// TIA Portal V17 export
// export: Created 2025-03-13T10:30:57.8594611Z, ExportSetting WithDefaults, DisplayName Totally Integrated Automation Portal, DisplayVersion V17 Update 8, DisplayName TIA Portal Openness, DisplayVersion V17 Update 8, DisplayName TIA Portal Version Control Interface, DisplayVersion V17, DisplayName SINAMICS Startdrive Advanced, DisplayVersion V17 SP2, DisplayName SINAMICS Startdrive G110M, G120, G120C, G120D, G120P, G115D, DisplayVersion V17 SP2, DisplayName SINAMICS Startdrive G130, G150, S120, S150, SINAMICS MV, S210, DisplayVersion V17 SP2, DisplayName STEP 7 Professional, DisplayVersion V17 Update 8, DisplayName SINUMERIK ONE STEP 7 Toolbox, DisplayVersion V17 Update 12, DisplayName SINUMERIK 840D sl STEP 7 Toolbox, DisplayVersion V17 Update 12, DisplayName STEP 7 Safety, DisplayVersion V17 Update 6, DisplayName WinCC Advanced, DisplayVersion V17 Update 8
DATA_BLOCK "DB505_HMI_SetUp"   // DB505
{ S7_Optimized_Access := 'FALSE'; DB_Accessible_From_OPC_UA := 'FALSE' }
AUTHOR : ETXETAR
VERSION : 1.0
// stored: AutoNumber false, DBAccessibleFromOPCUA false, DBAccessibleFromWebserver true, IsOnlyStoredInLoadMemory false, IsWriteProtectedInAS false
   VAR
      Setup1 : Struct
         Movement_EndPos : Struct   // Movement End Pos
            movement1EndPosLeft : Bool;   // Movement End Pos
            movement1EndPosRight : Bool;   // Movement End Pos
            movement2EndPosLeft : Bool;   // Movement End Pos
            movement2EndPosRight : Bool;   // Movement End Pos
            movement3EndPosLeft : Bool;   // Movement End Pos
            movement3EndPosRight : Bool;   // Movement End Pos
            movement4EndPosLeft : Bool;   // Movement End Pos
            movement4EndPosRight : Bool;   // Movement End Pos
            movement5EndPosLeft : Bool;   // Movement End Pos
            movement5EndPosRight : Bool;   // Movement End Pos
            movement6EndPosLeft : Bool;   // Movement End Pos
            movement6EndPosRight : Bool;   // Movement End Pos
            movement7EndPosLeft : Bool;   // Movement End Pos
            movement7EndPosRight : Bool;   // Movement End Pos
            movement8EndPosLeft : Bool;   // Movement End Pos
            movement8EndPosRight : Bool;   // Movement End Pos
            movement9EndPosLeft : Bool;   // Movement End Pos
            movement9EndPosRight : Bool;   // Movement End Pos
            movement10EndPosLeft : Bool;   // Movement End Pos
            movement10EndPosRight : Bool;   // Movement End Pos
            movement11EndPosLeft : Bool;   // Movement End Pos
            movement11EndPosRight : Bool;   // Movement End Pos
            movement12EndPosLeft : Bool;   // Movement End Pos
            movement12EndPosRight : Bool;   // Movement End Pos
            movement13EndPosLeft : Bool;   // Movement End Pos
            movement13EndPosRight : Bool;   // Movement End Pos
            movement14EndPosLeft : Bool;   // Movement End Pos
            movement14EndPosRight : Bool;   // Movement End Pos
            movement15EndPosLeft : Bool;   // Movement End Pos
            movement15EndPosRight : Bool;   // Movement End Pos
            movement16EndPosLeft : Bool;   // Movement End Pos
            movement16EndPosRight : Bool;   // Movement End Pos
            movement17EndPosLeft : Bool;   // Movement End Pos
            movement17EndPosRight : Bool;   // Movement End Pos
            movement18EndPosLeft : Bool;   // Movement End Pos
            movement18EndPosRight : Bool;   // Movement End Pos
            movement19EndPosLeft : Bool;   // Movement End Pos
            movement19EndPosRight : Bool;   // Movement End Pos
            movement20EndPosLeft : Bool;   // Movement End Pos
            movement20EndPosRight : Bool;   // Movement End Pos
            movement21EndPosLeft : Bool;   // Movement End Pos
            movement21EndPosRight : Bool;   // Movement End Pos
            movement22EndPosLeft : Bool;   // Movement End Pos
            movement22EndPosRight : Bool;   // Movement End Pos
            movement23EndPosLeft : Bool;   // Movement End Pos
            movement23EndPosRight : Bool;   // Movement End Pos
            movement24EndPosLeft : Bool;   // Movement End Pos
            movement24EndPosRight : Bool;   // Movement End Pos
            movement25EndPosLeft : Bool;   // Movement End Pos
            movement25EndPosRight : Bool;   // Movement End Pos
            movement26EndPosLeft : Bool;   // Movement End Pos
            movement26EndPosRight : Bool;   // Movement End Pos
            movement27EndPosLeft : Bool;   // Movement End Pos
            movement27EndPosRight : Bool;   // Movement End Pos
            movement28EndPosLeft : Bool;   // Movement End Pos
            movement28EndPosRight : Bool;   // Movement End Pos
            movement29EndPosLeft : Bool;   // Movement End Pos
            movement29EndPosRight : Bool;   // Movement End Pos
            movement30EndPosLeft : Bool;   // Movement End Pos
            movement30EndPosRight : Bool;   // Movement End Pos
            movement31EndPosLeft : Bool;   // Movement End Pos
            movement31EndPosRight : Bool;   // Movement End Pos
            movement32EndPosLeft : Bool;   // Movement End Pos
            movement32EndPosRight : Bool;   // Movement End Pos
            movement33EndPosLeft : Bool;   // Movement End Pos
            movement33EndPosRight : Bool;   // Movement End Pos
            movement34EndPosLeft : Bool;   // Movement End Pos
            movement34EndPosRight : Bool;   // Movement End Pos
            movement35EndPosLeft : Bool;   // Movement End Pos
            movement35EndPosRight : Bool;   // Movement End Pos
            movement36EndPosLeft : Bool;   // Movement End Pos
            movement36EndPosRight : Bool;   // Movement End Pos
            movement37EndPosLeft : Bool;   // Movement End Pos
            movement37EndPosRight : Bool;   // Movement End Pos
            movement38EndPosLeft : Bool;   // Movement End Pos
            movement38EndPosRight : Bool;   // Movement End Pos
            movement39EndPosLeft : Bool;   // Movement End Pos
            movement39EndPosRight : Bool;   // Movement End Pos
            movement40EndPosLeft : Bool;   // Movement End Pos
            movement40EndPosRight : Bool;   // Movement End Pos
            movement41EndPosLeft : Bool;   // Movement End Pos
            movement41EndPosRight : Bool;   // Movement End Pos
            movement42EndPosLeft : Bool;   // Movement End Pos
            movement42EndPosRight : Bool;   // Movement End Pos
            movement43EndPosLeft : Bool;   // Movement End Pos
            movement43EndPosRight : Bool;   // Movement End Pos
            movement44EndPosLeft : Bool;   // Movement End Pos
            movement44EndPosRight : Bool;   // Movement End Pos
            movement45EndPosLeft : Bool;   // Movement End Pos
            movement45EndPosRight : Bool;   // Movement End Pos
            movement46EndPosLeft : Bool;   // Movement End Pos
            movement46EndPosRight : Bool;   // Movement End Pos
            movement47EndPosLeft : Bool;   // Movement End Pos
            movement47EndPosRight : Bool;   // Movement End Pos
            movement48EndPosLeft : Bool;   // Movement End Pos
            movement48EndPosRight : Bool;   // Movement End Pos
            movement49EndPosLeft : Bool;   // Movement End Pos
            movement49EndPosRight : Bool;   // Movement End Pos
            movement50EndPosLeft : Bool;   // Movement End Pos
            movement50EndPosRight : Bool;   // Movement End Pos
            movement51EndPosLeft : Bool;   // Movement End Pos
            movement51EndPosRight : Bool;   // Movement End Pos
            movement52EndPosLeft : Bool;   // Movement End Pos
            movement52EndPosRight : Bool;   // Movement End Pos
            movement53EndPosLeft : Bool;   // Movement End Pos
            movement53EndPosRight : Bool;   // Movement End Pos
            movement54EndPosLeft : Bool;   // Movement End Pos
            movement54EndPosRight : Bool;   // Movement End Pos
            movement55EndPosLeft : Bool;   // Movement End Pos
            movement55EndPosRight : Bool;   // Movement End Pos
            movement56EndPosLeft : Bool;   // Movement End Pos
            movement56EndPosRight : Bool;   // Movement End Pos
            movement57EndPosLeft : Bool;   // Movement End Pos
            movement57EndPosRight : Bool;   // Movement End Pos
            movement58EndPosLeft : Bool;   // Movement End Pos
            movement58EndPosRight : Bool;   // Movement End Pos
            movement59EndPosLeft : Bool;   // Movement End Pos
            movement59EndPosRight : Bool;   // Movement End Pos
            movement60EndPosLeft : Bool;   // Movement End Pos
            movement60EndPosRight : Bool;   // Movement End Pos
            movement61EndPosLeft : Bool;   // Movement End Pos
            movement61EndPosRight : Bool;   // Movement End Pos
            movement62EndPosLeft : Bool;   // Movement End Pos
            movement62EndPosRight : Bool;   // Movement End Pos
            movement63EndPosLeft : Bool;   // Movement End Pos
            movement63EndPosRight : Bool;   // Movement End Pos
            movement64EndPosLeft : Bool;   // Movement End Pos
            movement64EndPosRight : Bool;   // Movement End Pos
            movement65EndPosLeft : Bool;   // Movement End Pos
            movement65EndPosRight : Bool;   // Movement End Pos
            movement66EndPosLeft : Bool;   // Movement End Pos
            movement66EndPosRight : Bool;   // Movement End Pos
            movement67EndPosLeft : Bool;   // Movement End Pos
            movement67EndPosRight : Bool;   // Movement End Pos
            movement68EndPosLeft : Bool;   // Movement End Pos
            movement68EndPosRight : Bool;   // Movement End Pos
            movement69EndPosLeft : Bool;   // Movement End Pos
            movement69EndPosRight : Bool;   // Movement End Pos
            movement70EndPosLeft : Bool;   // Movement End Pos
            movement70EndPosRight : Bool;   // Movement End Pos
            movement71EndPosLeft : Bool;   // Movement End Pos
            movement71EndPosRight : Bool;   // Movement End Pos
            movement72EndPosLeft : Bool;   // Movement End Pos
            movement72EndPosRight : Bool;   // Movement End Pos
            movement73EndPosLeft : Bool;   // Movement End Pos
            movement73EndPosRight : Bool;   // Movement End Pos
            movement74EndPosLeft : Bool;   // Movement End Pos
            movement74EndPosRight : Bool;   // Movement End Pos
            movement75EndPosLeft : Bool;   // Movement End Pos
            movement75EndPosRight : Bool;   // Movement End Pos
            movement76EndPosLeft : Bool;   // Movement End Pos
            movement76EndPosRight : Bool;   // Movement End Pos
            movement77EndPosLeft : Bool;   // Movement End Pos
            movement77EndPosRight : Bool;   // Movement End Pos
            movement78EndPosLeft : Bool;   // Movement End Pos
            movement78EndPosRight : Bool;   // Movement End Pos
            movement79EndPosLeft : Bool;   // Movement End Pos
            movement79EndPosRight : Bool;   // Movement End Pos
            movement80EndPosLeft : Bool;   // Movement End Pos
            movement80EndPosRight : Bool;   // Movement End Pos
            movement81EndPosLeft : Bool;   // Movement End Pos
            movement81EndPosRight : Bool;   // Movement End Pos
            movement82EndPosLeft : Bool;   // Movement End Pos
            movement82EndPosRight : Bool;   // Movement End Pos
            movement83EndPosLeft : Bool;   // Movement End Pos
            movement83EndPosRight : Bool;   // Movement End Pos
            movement84EndPosLeft : Bool;   // Movement End Pos
            movement84EndPosRight : Bool;   // Movement End Pos
            movement85EndPosLeft : Bool;   // Movement End Pos
            movement85EndPosRight : Bool;   // Movement End Pos
            movement86EndPosLeft : Bool;   // Movement End Pos
            movement86EndPosRight : Bool;   // Movement End Pos
            movement87EndPosLeft : Bool;   // Movement End Pos
            movement87EndPosRight : Bool;   // Movement End Pos
            movement88EndPosLeft : Bool;   // Movement End Pos
            movement88EndPosRight : Bool;   // Movement End Pos
            movement89EndPosLeft : Bool;   // Movement End Pos
            movement89EndPosRight : Bool;   // Movement End Pos
            movement90EndPosLeft : Bool;   // Movement End Pos
            movement90EndPosRight : Bool;   // Movement End Pos
            movement91EndPosLeft : Bool;   // Movement End Pos
            movement91EndPosRight : Bool;   // Movement End Pos
            movement92EndPosLeft : Bool;   // Movement End Pos
            movement92EndPosRight : Bool;   // Movement End Pos
            movement93EndPosLeft : Bool;   // Movement End Pos
            movement93EndPosRight : Bool;   // Movement End Pos
            movement94EndPosLeft : Bool;   // Movement End Pos
            movement94EndPosRight : Bool;   // Movement End Pos
            movement95EndPosLeft : Bool;   // Movement End Pos
            movement95EndPosRight : Bool;   // Movement End Pos
            movement96EndPosLeft : Bool;   // Movement End Pos
            movement96EndPosRight : Bool;   // Movement End Pos
            movement97EndPosLeft : Bool;   // Movement End Pos
            movement97EndPosRight : Bool;   // Movement End Pos
            movement98EndPosLeft : Bool;   // Movement End Pos
            movement98EndPosRight : Bool;   // Movement End Pos
            movement99EndPosLeft : Bool;   // Movement End Pos
            movement99EndPosRight : Bool;   // Movement End Pos
            movement100EndPosLeft : Bool;   // Movement End Pos
            movement100EndPosRight : Bool;   // Movement End Pos
            movement101EndPosLeft : Bool;   // Movement End Pos
            movement101EndPosRight : Bool;   // Movement End Pos
            movement102EndPosLeft : Bool;   // Movement End Pos
            movement102EndPosRight : Bool;   // Movement End Pos
            movement103EndPosLeft : Bool;   // Movement End Pos
            movement103EndPosRight : Bool;   // Movement End Pos
            movement104EndPosLeft : Bool;   // Movement End Pos
            movement104EndPosRight : Bool;   // Movement End Pos
            movement105EndPosLeft : Bool;   // Movement End Pos
            movement105EndPosRight : Bool;   // Movement End Pos
            movement106EndPosLeft : Bool;   // Movement End Pos
            movement106EndPosRight : Bool;   // Movement End Pos
            movement107EndPosLeft : Bool;   // Movement End Pos
            movement107EndPosRight : Bool;   // Movement End Pos
            movement108EndPosLeft : Bool;   // Movement End Pos
            movement108EndPosRight : Bool;   // Movement End Pos
            movement109EndPosLeft : Bool;   // Movement End Pos
            movement109EndPosRight : Bool;   // Movement End Pos
            movement110EndPosLeft : Bool;   // Movement End Pos
            movement110EndPosRight : Bool;   // Movement End Pos
            movement111EndPosLeft : Bool;   // Movement End Pos
            movement111EndPosRight : Bool;   // Movement End Pos
            movement112EndPosLeft : Bool;   // Movement End Pos
            movement112EndPosRight : Bool;   // Movement End Pos
            movement113EndPosLeft : Bool;   // Movement End Pos
            movement113EndPosRight : Bool;   // Movement End Pos
            movement114EndPosLeft : Bool;   // Movement End Pos
            movement114EndPosRight : Bool;   // Movement End Pos
            movement115EndPosLeft : Bool;   // Movement End Pos
            movement115EndPosRight : Bool;   // Movement End Pos
            movement116EndPosLeft : Bool;   // Movement End Pos
            movement116EndPosRight : Bool;   // Movement End Pos
            movement117EndPosLeft : Bool;   // Movement End Pos
            movement117EndPosRight : Bool;   // Movement End Pos
            movement118EndPosLeft : Bool;   // Movement End Pos
            movement118EndPosRight : Bool;   // Movement End Pos
            movement119EndPosLeft : Bool;   // Movement End Pos
            movement119EndPosRight : Bool;   // Movement End Pos
            movement120EndPosLeft : Bool;   // Movement End Pos
            movement120EndPosRight : Bool;   // Movement End Pos
            movement121EndPosLeft : Bool;   // Movement End Pos
            movement121EndPosRight : Bool;   // Movement End Pos
            movement122EndPosLeft : Bool;   // Movement End Pos
            movement122EndPosRight : Bool;   // Movement End Pos
            movement123EndPosLeft : Bool;   // Movement End Pos
            movement123EndPosRight : Bool;   // Movement End Pos
            movement124EndPosLeft : Bool;   // Movement End Pos
            movement124EndPosRight : Bool;   // Movement End Pos
            movement125EndPosLeft : Bool;   // Movement End Pos
            movement125EndPosRight : Bool;   // Movement End Pos
            movement126EndPosLeft : Bool;   // Movement End Pos
            movement126EndPosRight : Bool;   // Movement End Pos
            movement127EndPosLeft : Bool;   // Movement End Pos
            movement127EndPosRight : Bool;   // Movement End Pos
            movement128EndPosLeft : Bool;   // Movement End Pos
            movement128EndPosRight : Bool;   // Movement End Pos
            movement129EndPosLeft : Bool;   // Movement End Pos
            movement129EndPosRight : Bool;   // Movement End Pos
            movement130EndPosLeft : Bool;   // Movement End Pos
            movement130EndPosRight : Bool;   // Movement End Pos
            movement131EndPosLeft : Bool;   // Movement End Pos
            movement131EndPosRight : Bool;   // Movement End Pos
            movement132EndPosLeft : Bool;   // Movement End Pos
            movement132EndPosRight : Bool;   // Movement End Pos
            movement133EndPosLeft : Bool;   // Movement End Pos
            movement133EndPosRight : Bool;   // Movement End Pos
            movement134EndPosLeft : Bool;   // Movement End Pos
            movement134EndPosRight : Bool;   // Movement End Pos
            movement135EndPosLeft : Bool;   // Movement End Pos
            movement135EndPosRight : Bool;   // Movement End Pos
            movement136EndPosLeft : Bool;   // Movement End Pos
            movement136EndPosRight : Bool;   // Movement End Pos
            movement137EndPosLeft : Bool;   // Movement End Pos
            movement137EndPosRight : Bool;   // Movement End Pos
            movement138EndPosLeft : Bool;   // Movement End Pos
            movement138EndPosRight : Bool;   // Movement End Pos
            movement139EndPosLeft : Bool;   // Movement End Pos
            movement139EndPosRight : Bool;   // Movement End Pos
            movement140EndPosLeft : Bool;   // Movement End Pos
            movement140EndPosRight : Bool;   // Movement End Pos
            movement141EndPosLeft : Bool;   // Movement End Pos
            movement141EndPosRight : Bool;   // Movement End Pos
            movement142EndPosLeft : Bool;   // Movement End Pos
            movement142EndPosRight : Bool;   // Movement End Pos
            movement143EndPosLeft : Bool;   // Movement End Pos
            movement143EndPosRight : Bool;   // Movement End Pos
            movement144EndPosLeft : Bool;   // Movement End Pos
            movement144EndPosRight : Bool;   // Movement End Pos
            movement145EndPosLeft : Bool;   // Movement End Pos
            movement145EndPosRight : Bool;   // Movement End Pos
            movement146EndPosLeft : Bool;   // Movement End Pos
            movement146EndPosRight : Bool;   // Movement End Pos
            movement147EndPosLeft : Bool;   // Movement End Pos
            movement147EndPosRight : Bool;   // Movement End Pos
            movement148EndPosLeft : Bool;   // Movement End Pos
            movement148EndPosRight : Bool;   // Movement End Pos
            movement149EndPosLeft : Bool;   // Movement End Pos
            movement149EndPosRight : Bool;   // Movement End Pos
            movement150EndPosLeft : Bool;   // Movement End Pos
            movement150EndPosRight : Bool;   // Movement End Pos
            movement151EndPosLeft : Bool;   // Movement End Pos
            movement151EndPosRight : Bool;   // Movement End Pos
            movement152EndPosLeft : Bool;   // Movement End Pos
            movement152EndPosRight : Bool;   // Movement End Pos
            movement153EndPosLeft : Bool;   // Movement End Pos
            movement153EndPosRight : Bool;   // Movement End Pos
            movement154EndPosLeft : Bool;   // Movement End Pos
            movement154EndPosRight : Bool;   // Movement End Pos
            movement155EndPosLeft : Bool;   // Movement End Pos
            movement155EndPosRight : Bool;   // Movement End Pos
            movement156EndPosLeft : Bool;   // Movement End Pos
            movement156EndPosRight : Bool;   // Movement End Pos
            movement157EndPosLeft : Bool;   // Movement End Pos
            movement157EndPosRight : Bool;   // Movement End Pos
            movement158EndPosLeft : Bool;   // Movement End Pos
            movement158EndPosRight : Bool;   // Movement End Pos
            movement159EndPosLeft : Bool;   // Movement End Pos
            movement159EndPosRight : Bool;   // Movement End Pos
            movement160EndPosLeft : Bool;   // Movement End Pos
            movement160EndPosRight : Bool;   // Movement End Pos
            movement161EndPosLeft : Bool;   // Movement End Pos
            movement161EndPosRight : Bool;   // Movement End Pos
            movement162EndPosLeft : Bool;   // Movement End Pos
            movement162EndPosRight : Bool;   // Movement End Pos
            movement163EndPosLeft : Bool;   // Movement End Pos
            movement163EndPosRight : Bool;   // Movement End Pos
            movement164EndPosLeft : Bool;   // Movement End Pos
            movement164EndPosRight : Bool;   // Movement End Pos
            movement165EndPosLeft : Bool;   // Movement End Pos
            movement165EndPosRight : Bool;   // Movement End Pos
            movement166EndPosLeft : Bool;   // Movement End Pos
            movement166EndPosRight : Bool;   // Movement End Pos
            movement167EndPosLeft : Bool;   // Movement End Pos
            movement167EndPosRight : Bool;   // Movement End Pos
            movement168EndPosLeft : Bool;   // Movement End Pos
            movement168EndPosRight : Bool;   // Movement End Pos
            movement169EndPosLeft : Bool;   // Movement End Pos
            movement169EndPosRight : Bool;   // Movement End Pos
            movement170EndPosLeft : Bool;   // Movement End Pos
            movement170EndPosRight : Bool;   // Movement End Pos
            movement171EndPosLeft : Bool;   // Movement End Pos
            movement171EndPosRight : Bool;   // Movement End Pos
            movement172EndPosLeft : Bool;   // Movement End Pos
            movement172EndPosRight : Bool;   // Movement End Pos
            movement173EndPosLeft : Bool;   // Movement End Pos
            movement173EndPosRight : Bool;   // Movement End Pos
            movement174EndPosLeft : Bool;   // Movement End Pos
            movement174EndPosRight : Bool;   // Movement End Pos
            movement175EndPosLeft : Bool;   // Movement End Pos
            movement175EndPosRight : Bool;   // Movement End Pos
            movement176EndPosLeft : Bool;   // Movement End Pos
            movement176EndPosRight : Bool;   // Movement End Pos
            movement177EndPosLeft : Bool;   // Movement End Pos
            movement177EndPosRight : Bool;   // Movement End Pos
            movement178EndPosLeft : Bool;   // Movement End Pos
            movement178EndPosRight : Bool;   // Movement End Pos
            movement179EndPosLeft : Bool;   // Movement End Pos
            movement179EndPosRight : Bool;   // Movement End Pos
            movement180EndPosLeft : Bool;   // Movement End Pos
            movement180EndPosRight : Bool;   // Movement End Pos
            movement181EndPosLeft : Bool;   // Movement End Pos
            movement181EndPosRight : Bool;   // Movement End Pos
            movement182EndPosLeft : Bool;   // Movement End Pos
            movement182EndPosRight : Bool;   // Movement End Pos
            movement183EndPosLeft : Bool;   // Movement End Pos
            movement183EndPosRight : Bool;   // Movement End Pos
            movement184EndPosLeft : Bool;   // Movement End Pos
            movement184EndPosRight : Bool;   // Movement End Pos
            movement185EndPosLeft : Bool;   // Movement End Pos
            movement185EndPosRight : Bool;   // Movement End Pos
            movement186EndPosLeft : Bool;   // Movement End Pos
            movement186EndPosRight : Bool;   // Movement End Pos
            movement187EndPosLeft : Bool;   // Movement End Pos
            movement187EndPosRight : Bool;   // Movement End Pos
            movement188EndPosLeft : Bool;   // Movement End Pos
            movement188EndPosRight : Bool;   // Movement End Pos
            movement189EndPosLeft : Bool;   // Movement End Pos
            movement189EndPosRight : Bool;   // Movement End Pos
            movement190EndPosLeft : Bool;   // Movement End Pos
            movement190EndPosRight : Bool;   // Movement End Pos
            movement191EndPosLeft : Bool;   // Movement End Pos
            movement191EndPosRight : Bool;   // Movement End Pos
            movement192EndPosLeft : Bool;   // Movement End Pos
            movement192EndPosRight : Bool;   // Movement End Pos
            movement193EndPosLeft : Bool;   // Movement End Pos
            movement193EndPosRight : Bool;   // Movement End Pos
            movement194EndPosLeft : Bool;   // Movement End Pos
            movement194EndPosRight : Bool;   // Movement End Pos
            movement195EndPosLeft : Bool;   // Movement End Pos
            movement195EndPosRight : Bool;   // Movement End Pos
            movement196EndPosLeft : Bool;   // Movement End Pos
            movement196EndPosRight : Bool;   // Movement End Pos
            movement197EndPosLeft : Bool;   // Movement End Pos
            movement197EndPosRight : Bool;   // Movement End Pos
            movement198EndPosLeft : Bool;   // Movement End Pos
            movement198EndPosRight : Bool;   // Movement End Pos
            movement199EndPosLeft : Bool;   // Movement End Pos
            movement199EndPosRight : Bool;   // Movement End Pos
            movement200EndPosLeft : Bool;   // Movement End Pos
            movement200EndPosRight : Bool;   // Movement End Pos
            movement201EndPosLeft : Bool;   // Movement End Pos
            movement201EndPosRight : Bool;   // Movement End Pos
            movement202EndPosLeft : Bool;   // Movement End Pos
            movement202EndPosRight : Bool;   // Movement End Pos
            movement203EndPosLeft : Bool;   // Movement End Pos
            movement203EndPosRight : Bool;   // Movement End Pos
            movement204EndPosLeft : Bool;   // Movement End Pos
            movement204EndPosRight : Bool;   // Movement End Pos
            movement205EndPosLeft : Bool;   // Movement End Pos
            movement205EndPosRight : Bool;   // Movement End Pos
            movement206EndPosLeft : Bool;   // Movement End Pos
            movement206EndPosRight : Bool;   // Movement End Pos
            movement207EndPosLeft : Bool;   // Movement End Pos
            movement207EndPosRight : Bool;   // Movement End Pos
            movement208EndPosLeft : Bool;   // Movement End Pos
            movement208EndPosRight : Bool;   // Movement End Pos
            movement209EndPosLeft : Bool;   // Movement End Pos
            movement209EndPosRight : Bool;   // Movement End Pos
            movement210EndPosLeft : Bool;   // Movement End Pos
            movement210EndPosRight : Bool;   // Movement End Pos
            movement211EndPosLeft : Bool;   // Movement End Pos
            movement211EndPosRight : Bool;   // Movement End Pos
            movement212EndPosLeft : Bool;   // Movement End Pos
            movement212EndPosRight : Bool;   // Movement End Pos
            movement213EndPosLeft : Bool;   // Movement End Pos
            movement213EndPosRight : Bool;   // Movement End Pos
            movement214EndPosLeft : Bool;   // Movement End Pos
            movement214EndPosRight : Bool;   // Movement End Pos
            movement215EndPosLeft : Bool;   // Movement End Pos
            movement215EndPosRight : Bool;   // Movement End Pos
            movement216EndPosLeft : Bool;   // Movement End Pos
            movement216EndPosRight : Bool;   // Movement End Pos
            movement217EndPosLeft : Bool;   // Movement End Pos
            movement217EndPosRight : Bool;   // Movement End Pos
            movement218EndPosLeft : Bool;   // Movement End Pos
            movement218EndPosRight : Bool;   // Movement End Pos
            movement219EndPosLeft : Bool;   // Movement End Pos
            movement219EndPosRight : Bool;   // Movement End Pos
            movement220EndPosLeft : Bool;   // Movement End Pos
            movement220EndPosRight : Bool;   // Movement End Pos
            movement221EndPosLeft : Bool;   // Movement End Pos
            movement221EndPosRight : Bool;   // Movement End Pos
            movement222EndPosLeft : Bool;   // Movement End Pos
            movement222EndPosRight : Bool;   // Movement End Pos
            movement223EndPosLeft : Bool;   // Movement End Pos
            movement223EndPosRight : Bool;   // Movement End Pos
            movement224EndPosLeft : Bool;   // Movement End Pos
            movement224EndPosRight : Bool;   // Movement End Pos
            movement225EndPosLeft : Bool;   // Movement End Pos
            movement225EndPosRight : Bool;   // Movement End Pos
            movement226EndPosLeft : Bool;   // Movement End Pos
            movement226EndPosRight : Bool;   // Movement End Pos
            movement227EndPosLeft : Bool;   // Movement End Pos
            movement227EndPosRight : Bool;   // Movement End Pos
            movement228EndPosLeft : Bool;   // Movement End Pos
            movement228EndPosRight : Bool;   // Movement End Pos
            movement229EndPosLeft : Bool;   // Movement End Pos
            movement229EndPosRight : Bool;   // Movement End Pos
            movement230EndPosLeft : Bool;   // Movement End Pos
            movement230EndPosRight : Bool;   // Movement End Pos
            movement231EndPosLeft : Bool;   // Movement End Pos
            movement231EndPosRight : Bool;   // Movement End Pos
            movement232EndPosLeft : Bool;   // Movement End Pos
            movement232EndPosRight : Bool;   // Movement End Pos
            movement233EndPosLeft : Bool;   // Movement End Pos
            movement233EndPosRight : Bool;   // Movement End Pos
            movement234EndPosLeft : Bool;   // Movement End Pos
            movement234EndPosRight : Bool;   // Movement End Pos
            movement235EndPosLeft : Bool;   // Movement End Pos
            movement235EndPosRight : Bool;   // Movement End Pos
            movement236EndPosLeft : Bool;   // Movement End Pos
            movement236EndPosRight : Bool;   // Movement End Pos
            movement237EndPosLeft : Bool;   // Movement End Pos
            movement237EndPosRight : Bool;   // Movement End Pos
            movement238EndPosLeft : Bool;   // Movement End Pos
            movement238EndPosRight : Bool;   // Movement End Pos
            movement239EndPosLeft : Bool;   // Movement End Pos
            movement239EndPosRight : Bool;   // Movement End Pos
            movement240EndPosLeft : Bool;   // Movement End Pos
            movement240EndPosRight : Bool;   // Movement End Pos
            movement241EndPosLeft : Bool;   // Movement End Pos
            movement241EndPosRight : Bool;   // Movement End Pos
            movement242EndPosLeft : Bool;   // Movement End Pos
            movement242EndPosRight : Bool;   // Movement End Pos
            movement243EndPosLeft : Bool;   // Movement End Pos
            movement243EndPosRight : Bool;   // Movement End Pos
            movement244EndPosLeft : Bool;   // Movement End Pos
            movement244EndPosRight : Bool;   // Movement End Pos
            movement245EndPosLeft : Bool;   // Movement End Pos
            movement245EndPosRight : Bool;   // Movement End Pos
            movement246EndPosLeft : Bool;   // Movement End Pos
            movement246EndPosRight : Bool;   // Movement End Pos
            movement247EndPosLeft : Bool;   // Movement End Pos
            movement247EndPosRight : Bool;   // Movement End Pos
            movement248EndPosLeft : Bool;   // Movement End Pos
            movement248EndPosRight : Bool;   // Movement End Pos
            movement249EndPosLeft : Bool;   // Movement End Pos
            movement249EndPosRight : Bool;   // Movement End Pos
            movement250EndPosLeft : Bool;   // Movement End Pos
            movement250EndPosRight : Bool;   // Movement End Pos
            movement251EndPosLeft : Bool;   // Movement End Pos
            movement251EndPosRight : Bool;   // Movement End Pos
            movement252EndPosLeft : Bool;   // Movement End Pos
            movement252EndPosRight : Bool;   // Movement End Pos
            movement253EndPosLeft : Bool;   // Movement End Pos
            movement253EndPosRight : Bool;   // Movement End Pos
            movement254EndPosLeft : Bool;   // Movement End Pos
            movement254EndPosRight : Bool;   // Movement End Pos
            movement255EndPosLeft : Bool;   // Movement End Pos
            movement255EndPosRight : Bool;   // Movement End Pos
            movement256EndPosLeft : Bool;   // Movement End Pos
            movement256EndPosRight : Bool;   // Movement End Pos
         END_STRUCT;
         Movement_Executability : Struct   // Movement Executability
            movement1ExecutabilityLeft : Bool;   // Movement Executability
            movement1ExecutabilityRight : Bool;   // Movement Executability
            movement2ExecutabilityLeft : Bool;   // Movement Executability
            movement2ExecutabilityRight : Bool;   // Movement Executability
            movement3ExecutabilityLeft : Bool;   // Movement Executability
            movement3ExecutabilityRight : Bool;   // Movement Executability
            movement4ExecutabilityLeft : Bool;   // Movement Executability
            movement4ExecutabilityRight : Bool;   // Movement Executability
            movement5ExecutabilityLeft : Bool;   // Movement Executability
            movement5ExecutabilityRight : Bool;   // Movement Executability
            movement6ExecutabilityLeft : Bool;   // Movement Executability
            movement6ExecutabilityRight : Bool;   // Movement Executability
            movement7ExecutabilityLeft : Bool;   // Movement Executability
            movement7ExecutabilityRight : Bool;   // Movement Executability
            movement8ExecutabilityLeft : Bool;   // Movement Executability
            movement8ExecutabilityRight : Bool;   // Movement Executability
            movement9ExecutabilityLeft : Bool;   // Movement Executability
            movement9ExecutabilityRight : Bool;   // Movement Executability
            movement10ExecutabilityLeft : Bool;   // Movement Executability
            movement10ExecutabilityRight : Bool;   // Movement Executability
            movement11ExecutabilityLeft : Bool;   // Movement Executability
            movement11ExecutabilityRight : Bool;   // Movement Executability
            movement12ExecutabilityLeft : Bool;   // Movement Executability
            movement12ExecutabilityRight : Bool;   // Movement Executability
            movement13ExecutabilityLeft : Bool;   // Movement Executability
            movement13ExecutabilityRight : Bool;   // Movement Executability
            movement14ExecutabilityLeft : Bool;   // Movement Executability
            movement14ExecutabilityRight : Bool;   // Movement Executability
            movement15ExecutabilityLeft : Bool;   // Movement Executability
            movement15ExecutabilityRight : Bool;   // Movement Executability
            movement16ExecutabilityLeft : Bool;   // Movement Executability
            movement16ExecutabilityRight : Bool;   // Movement Executability
            movement17ExecutabilityLeft : Bool;   // Movement Executability
            movement17ExecutabilityRight : Bool;   // Movement Executability
            movement18ExecutabilityLeft : Bool;   // Movement Executability
            movement18ExecutabilityRight : Bool;   // Movement Executability
            movement19ExecutabilityLeft : Bool;   // Movement Executability
            movement19ExecutabilityRight : Bool;   // Movement Executability
            movement20ExecutabilityLeft : Bool;   // Movement Executability
            movement20ExecutabilityRight : Bool;   // Movement Executability
            movement21ExecutabilityLeft : Bool;   // Movement Executability
            movement21ExecutabilityRight : Bool;   // Movement Executability
            movement22ExecutabilityLeft : Bool;   // Movement Executability
            movement22ExecutabilityRight : Bool;   // Movement Executability
            movement23ExecutabilityLeft : Bool;   // Movement Executability
            movement23ExecutabilityRight : Bool;   // Movement Executability
            movement24ExecutabilityLeft : Bool;   // Movement Executability
            movement24ExecutabilityRight : Bool;   // Movement Executability
            movement25ExecutabilityLeft : Bool;   // Movement Executability
            movement25ExecutabilityRight : Bool;   // Movement Executability
            movement26ExecutabilityLeft : Bool;   // Movement Executability
            movement26ExecutabilityRight : Bool;   // Movement Executability
            movement27ExecutabilityLeft : Bool;   // Movement Executability
            movement27ExecutabilityRight : Bool;   // Movement Executability
            movement28ExecutabilityLeft : Bool;   // Movement Executability
            movement28ExecutabilityRight : Bool;   // Movement Executability
            movement29ExecutabilityLeft : Bool;   // Movement Executability
            movement29ExecutabilityRight : Bool;   // Movement Executability
            movement30ExecutabilityLeft : Bool;   // Movement Executability
            movement30ExecutabilityRight : Bool;   // Movement Executability
            movement31ExecutabilityLeft : Bool;   // Movement Executability
            movement31ExecutabilityRight : Bool;   // Movement Executability
            movement32ExecutabilityLeft : Bool;   // Movement Executability
            movement32ExecutabilityRight : Bool;   // Movement Executability
            movement33ExecutabilityLeft : Bool;   // Movement Executability
            movement33ExecutabilityRight : Bool;   // Movement Executability
            movement34ExecutabilityLeft : Bool;   // Movement Executability
            movement34ExecutabilityRight : Bool;   // Movement Executability
            movement35ExecutabilityLeft : Bool;   // Movement Executability
            movement35ExecutabilityRight : Bool;   // Movement Executability
            movement36ExecutabilityLeft : Bool;   // Movement Executability
            movement36ExecutabilityRight : Bool;   // Movement Executability
            movement37ExecutabilityLeft : Bool;   // Movement Executability
            movement37ExecutabilityRight : Bool;   // Movement Executability
            movement38ExecutabilityLeft : Bool;   // Movement Executability
            movement38ExecutabilityRight : Bool;   // Movement Executability
            movement39ExecutabilityLeft : Bool;   // Movement Executability
            movement39ExecutabilityRight : Bool;   // Movement Executability
            movement40ExecutabilityLeft : Bool;   // Movement Executability
            movement40ExecutabilityRight : Bool;   // Movement Executability
            movement41ExecutabilityLeft : Bool;   // Movement Executability
            movement41ExecutabilityRight : Bool;   // Movement Executability
            movement42ExecutabilityLeft : Bool;   // Movement Executability
            movement42ExecutabilityRight : Bool;   // Movement Executability
            movement43ExecutabilityLeft : Bool;   // Movement Executability
            movement43ExecutabilityRight : Bool;   // Movement Executability
            movement44ExecutabilityLeft : Bool;   // Movement Executability
            movement44ExecutabilityRight : Bool;   // Movement Executability
            movement45ExecutabilityLeft : Bool;   // Movement Executability
            movement45ExecutabilityRight : Bool;   // Movement Executability
            movement46ExecutabilityLeft : Bool;   // Movement Executability
            movement46ExecutabilityRight : Bool;   // Movement Executability
            movement47ExecutabilityLeft : Bool;   // Movement Executability
            movement47ExecutabilityRight : Bool;   // Movement Executability
            movement48ExecutabilityLeft : Bool;   // Movement Executability
            movement48ExecutabilityRight : Bool;   // Movement Executability
            movement49ExecutabilityLeft : Bool;   // Movement Executability
            movement49ExecutabilityRight : Bool;   // Movement Executability
            movement50ExecutabilityLeft : Bool;   // Movement Executability
            movement50ExecutabilityRight : Bool;   // Movement Executability
            movement51ExecutabilityLeft : Bool;   // Movement Executability
            movement51ExecutabilityRight : Bool;   // Movement Executability
            movement52ExecutabilityLeft : Bool;   // Movement Executability
            movement52ExecutabilityRight : Bool;   // Movement Executability
            movement53ExecutabilityLeft : Bool;   // Movement Executability
            movement53ExecutabilityRight : Bool;   // Movement Executability
            movement54ExecutabilityLeft : Bool;   // Movement Executability
            movement54ExecutabilityRight : Bool;   // Movement Executability
            movement55ExecutabilityLeft : Bool;   // Movement Executability
            movement55ExecutabilityRight : Bool;   // Movement Executability
            movement56ExecutabilityLeft : Bool;   // Movement Executability
            movement56ExecutabilityRight : Bool;   // Movement Executability
            movement57ExecutabilityLeft : Bool;   // Movement Executability
            movement57ExecutabilityRight : Bool;   // Movement Executability
            movement58ExecutabilityLeft : Bool;   // Movement Executability
            movement58ExecutabilityRight : Bool;   // Movement Executability
            movement59ExecutabilityLeft : Bool;   // Movement Executability
            movement59ExecutabilityRight : Bool;   // Movement Executability
            movement60ExecutabilityLeft : Bool;   // Movement Executability
            movement60ExecutabilityRight : Bool;   // Movement Executability
            movement61ExecutabilityLeft : Bool;   // Movement Executability
            movement61ExecutabilityRight : Bool;   // Movement Executability
            movement62ExecutabilityLeft : Bool;   // Movement Executability
            movement62ExecutabilityRight : Bool;   // Movement Executability
            movement63ExecutabilityLeft : Bool;   // Movement Executability
            movement63ExecutabilityRight : Bool;   // Movement Executability
            movement64ExecutabilityLeft : Bool;   // Movement Executability
            movement64ExecutabilityRight : Bool;   // Movement Executability
            movement65ExecutabilityLeft : Bool;   // Movement Executability
            movement65ExecutabilityRight : Bool;   // Movement Executability
            movement66ExecutabilityLeft : Bool;   // Movement Executability
            movement66ExecutabilityRight : Bool;   // Movement Executability
            movement67ExecutabilityLeft : Bool;   // Movement Executability
            movement67ExecutabilityRight : Bool;   // Movement Executability
            movement68ExecutabilityLeft : Bool;   // Movement Executability
            movement68ExecutabilityRight : Bool;   // Movement Executability
            movement69ExecutabilityLeft : Bool;   // Movement Executability
            movement69ExecutabilityRight : Bool;   // Movement Executability
            movement70ExecutabilityLeft : Bool;   // Movement Executability
            movement70ExecutabilityRight : Bool;   // Movement Executability
            movement71ExecutabilityLeft : Bool;   // Movement Executability
            movement71ExecutabilityRight : Bool;   // Movement Executability
            movement72ExecutabilityLeft : Bool;   // Movement Executability
            movement72ExecutabilityRight : Bool;   // Movement Executability
            movement73ExecutabilityLeft : Bool;   // Movement Executability
            movement73ExecutabilityRight : Bool;   // Movement Executability
            movement74ExecutabilityLeft : Bool;   // Movement Executability
            movement74ExecutabilityRight : Bool;   // Movement Executability
            movement75ExecutabilityLeft : Bool;   // Movement Executability
            movement75ExecutabilityRight : Bool;   // Movement Executability
            movement76ExecutabilityLeft : Bool;   // Movement Executability
            movement76ExecutabilityRight : Bool;   // Movement Executability
            movement77ExecutabilityLeft : Bool;   // Movement Executability
            movement77ExecutabilityRight : Bool;   // Movement Executability
            movement78ExecutabilityLeft : Bool;   // Movement Executability
            movement78ExecutabilityRight : Bool;   // Movement Executability
            movement79ExecutabilityLeft : Bool;   // Movement Executability
            movement79ExecutabilityRight : Bool;   // Movement Executability
            movement80ExecutabilityLeft : Bool;   // Movement Executability
            movement80ExecutabilityRight : Bool;   // Movement Executability
            movement81ExecutabilityLeft : Bool;   // Movement Executability
            movement81ExecutabilityRight : Bool;   // Movement Executability
            movement82ExecutabilityLeft : Bool;   // Movement Executability
            movement82ExecutabilityRight : Bool;   // Movement Executability
            movement83ExecutabilityLeft : Bool;   // Movement Executability
            movement83ExecutabilityRight : Bool;   // Movement Executability
            movement84ExecutabilityLeft : Bool;   // Movement Executability
            movement84ExecutabilityRight : Bool;   // Movement Executability
            movement85ExecutabilityLeft : Bool;   // Movement Executability
            movement85ExecutabilityRight : Bool;   // Movement Executability
            movement86ExecutabilityLeft : Bool;   // Movement Executability
            movement86ExecutabilityRight : Bool;   // Movement Executability
            movement87ExecutabilityLeft : Bool;   // Movement Executability
            movement87ExecutabilityRight : Bool;   // Movement Executability
            movement88ExecutabilityLeft : Bool;   // Movement Executability
            movement88ExecutabilityRight : Bool;   // Movement Executability
            movement89ExecutabilityLeft : Bool;   // Movement Executability
            movement89ExecutabilityRight : Bool;   // Movement Executability
            movement90ExecutabilityLeft : Bool;   // Movement Executability
            movement90ExecutabilityRight : Bool;   // Movement Executability
            movement91ExecutabilityLeft : Bool;   // Movement Executability
            movement91ExecutabilityRight : Bool;   // Movement Executability
            movement92ExecutabilityLeft : Bool;   // Movement Executability
            movement92ExecutabilityRight : Bool;   // Movement Executability
            movement93ExecutabilityLeft : Bool;   // Movement Executability
            movement93ExecutabilityRight : Bool;   // Movement Executability
            movement94ExecutabilityLeft : Bool;   // Movement Executability
            movement94ExecutabilityRight : Bool;   // Movement Executability
            movement95ExecutabilityLeft : Bool;   // Movement Executability
            movement95ExecutabilityRight : Bool;   // Movement Executability
            movement96ExecutabilityLeft : Bool;   // Movement Executability
            movement96ExecutabilityRight : Bool;   // Movement Executability
            movement97ExecutabilityLeft : Bool;   // Movement Executability
            movement97ExecutabilityRight : Bool;   // Movement Executability
            movement98ExecutabilityLeft : Bool;   // Movement Executability
            movement98ExecutabilityRight : Bool;   // Movement Executability
            movement99ExecutabilityLeft : Bool;   // Movement Executability
            movement99ExecutabilityRight : Bool;   // Movement Executability
            movement100ExecutabilityLeft : Bool;   // Movement Executability
            movement100ExecutabilityRight : Bool;   // Movement Executability
            movement101ExecutabilityLeft : Bool;   // Movement Executability
            movement101ExecutabilityRight : Bool;   // Movement Executability
            movement102ExecutabilityLeft : Bool;   // Movement Executability
            movement102ExecutabilityRight : Bool;   // Movement Executability
            movement103ExecutabilityLeft : Bool;   // Movement Executability
            movement103ExecutabilityRight : Bool;   // Movement Executability
            movement104ExecutabilityLeft : Bool;   // Movement Executability
            movement104ExecutabilityRight : Bool;   // Movement Executability
            movement105ExecutabilityLeft : Bool;   // Movement Executability
            movement105ExecutabilityRight : Bool;   // Movement Executability
            movement106ExecutabilityLeft : Bool;   // Movement Executability
            movement106ExecutabilityRight : Bool;   // Movement Executability
            movement107ExecutabilityLeft : Bool;   // Movement Executability
            movement107ExecutabilityRight : Bool;   // Movement Executability
            movement108ExecutabilityLeft : Bool;   // Movement Executability
            movement108ExecutabilityRight : Bool;   // Movement Executability
            movement109ExecutabilityLeft : Bool;   // Movement Executability
            movement109ExecutabilityRight : Bool;   // Movement Executability
            movement110ExecutabilityLeft : Bool;   // Movement Executability
            movement110ExecutabilityRight : Bool;   // Movement Executability
            movement111ExecutabilityLeft : Bool;   // Movement Executability
            movement111ExecutabilityRight : Bool;   // Movement Executability
            movement112ExecutabilityLeft : Bool;   // Movement Executability
            movement112ExecutabilityRight : Bool;   // Movement Executability
            movement113ExecutabilityLeft : Bool;   // Movement Executability
            movement113ExecutabilityRight : Bool;   // Movement Executability
            movement114ExecutabilityLeft : Bool;   // Movement Executability
            movement114ExecutabilityRight : Bool;   // Movement Executability
            movement115ExecutabilityLeft : Bool;   // Movement Executability
            movement115ExecutabilityRight : Bool;   // Movement Executability
            movement116ExecutabilityLeft : Bool;   // Movement Executability
            movement116ExecutabilityRight : Bool;   // Movement Executability
            movement117ExecutabilityLeft : Bool;   // Movement Executability
            movement117ExecutabilityRight : Bool;   // Movement Executability
            movement118ExecutabilityLeft : Bool;   // Movement Executability
            movement118ExecutabilityRight : Bool;   // Movement Executability
            movement119ExecutabilityLeft : Bool;   // Movement Executability
            movement119ExecutabilityRight : Bool;   // Movement Executability
            movement120ExecutabilityLeft : Bool;   // Movement Executability
            movement120ExecutabilityRight : Bool;   // Movement Executability
            movement121ExecutabilityLeft : Bool;   // Movement Executability
            movement121ExecutabilityRight : Bool;   // Movement Executability
            movement122ExecutabilityLeft : Bool;   // Movement Executability
            movement122ExecutabilityRight : Bool;   // Movement Executability
            movement123ExecutabilityLeft : Bool;   // Movement Executability
            movement123ExecutabilityRight : Bool;   // Movement Executability
            movement124ExecutabilityLeft : Bool;   // Movement Executability
            movement124ExecutabilityRight : Bool;   // Movement Executability
            movement125ExecutabilityLeft : Bool;   // Movement Executability
            movement125ExecutabilityRight : Bool;   // Movement Executability
            movement126ExecutabilityLeft : Bool;   // Movement Executability
            movement126ExecutabilityRight : Bool;   // Movement Executability
            movement127ExecutabilityLeft : Bool;   // Movement Executability
            movement127ExecutabilityRight : Bool;   // Movement Executability
            movement128ExecutabilityLeft : Bool;   // Movement Executability
            movement128ExecutabilityRight : Bool;   // Movement Executability
            movement129ExecutabilityLeft : Bool;   // Movement Executability
            movement129ExecutabilityRight : Bool;   // Movement Executability
            movement130ExecutabilityLeft : Bool;   // Movement Executability
            movement130ExecutabilityRight : Bool;   // Movement Executability
            movement131ExecutabilityLeft : Bool;   // Movement Executability
            movement131ExecutabilityRight : Bool;   // Movement Executability
            movement132ExecutabilityLeft : Bool;   // Movement Executability
            movement132ExecutabilityRight : Bool;   // Movement Executability
            movement133ExecutabilityLeft : Bool;   // Movement Executability
            movement133ExecutabilityRight : Bool;   // Movement Executability
            movement134ExecutabilityLeft : Bool;   // Movement Executability
            movement134ExecutabilityRight : Bool;   // Movement Executability
            movement135ExecutabilityLeft : Bool;   // Movement Executability
            movement135ExecutabilityRight : Bool;   // Movement Executability
            movement136ExecutabilityLeft : Bool;   // Movement Executability
            movement136ExecutabilityRight : Bool;   // Movement Executability
            movement137ExecutabilityLeft : Bool;   // Movement Executability
            movement137ExecutabilityRight : Bool;   // Movement Executability
            movement138ExecutabilityLeft : Bool;   // Movement Executability
            movement138ExecutabilityRight : Bool;   // Movement Executability
            movement139ExecutabilityLeft : Bool;   // Movement Executability
            movement139ExecutabilityRight : Bool;   // Movement Executability
            movement140ExecutabilityLeft : Bool;   // Movement Executability
            movement140ExecutabilityRight : Bool;   // Movement Executability
            movement141ExecutabilityLeft : Bool;   // Movement Executability
            movement141ExecutabilityRight : Bool;   // Movement Executability
            movement142ExecutabilityLeft : Bool;   // Movement Executability
            movement142ExecutabilityRight : Bool;   // Movement Executability
            movement143ExecutabilityLeft : Bool;   // Movement Executability
            movement143ExecutabilityRight : Bool;   // Movement Executability
            movement144ExecutabilityLeft : Bool;   // Movement Executability
            movement144ExecutabilityRight : Bool;   // Movement Executability
            movement145ExecutabilityLeft : Bool;   // Movement Executability
            movement145ExecutabilityRight : Bool;   // Movement Executability
            movement146ExecutabilityLeft : Bool;   // Movement Executability
            movement146ExecutabilityRight : Bool;   // Movement Executability
            movement147ExecutabilityLeft : Bool;   // Movement Executability
            movement147ExecutabilityRight : Bool;   // Movement Executability
            movement148ExecutabilityLeft : Bool;   // Movement Executability
            movement148ExecutabilityRight : Bool;   // Movement Executability
            movement149ExecutabilityLeft : Bool;   // Movement Executability
            movement149ExecutabilityRight : Bool;   // Movement Executability
            movement150ExecutabilityLeft : Bool;   // Movement Executability
            movement150ExecutabilityRight : Bool;   // Movement Executability
            movement151ExecutabilityLeft : Bool;   // Movement Executability
            movement151ExecutabilityRight : Bool;   // Movement Executability
            movement152ExecutabilityLeft : Bool;   // Movement Executability
            movement152ExecutabilityRight : Bool;   // Movement Executability
            movement153ExecutabilityLeft : Bool;   // Movement Executability
            movement153ExecutabilityRight : Bool;   // Movement Executability
            movement154ExecutabilityLeft : Bool;   // Movement Executability
            movement154ExecutabilityRight : Bool;   // Movement Executability
            movement155ExecutabilityLeft : Bool;   // Movement Executability
            movement155ExecutabilityRight : Bool;   // Movement Executability
            movement156ExecutabilityLeft : Bool;   // Movement Executability
            movement156ExecutabilityRight : Bool;   // Movement Executability
            movement157ExecutabilityLeft : Bool;   // Movement Executability
            movement157ExecutabilityRight : Bool;   // Movement Executability
            movement158ExecutabilityLeft : Bool;   // Movement Executability
            movement158ExecutabilityRight : Bool;   // Movement Executability
            movement159ExecutabilityLeft : Bool;   // Movement Executability
            movement159ExecutabilityRight : Bool;   // Movement Executability
            movement160ExecutabilityLeft : Bool;   // Movement Executability
            movement160ExecutabilityRight : Bool;   // Movement Executability
            movement161ExecutabilityLeft : Bool;   // Movement Executability
            movement161ExecutabilityRight : Bool;   // Movement Executability
            movement162ExecutabilityLeft : Bool;   // Movement Executability
            movement162ExecutabilityRight : Bool;   // Movement Executability
            movement163ExecutabilityLeft : Bool;   // Movement Executability
            movement163ExecutabilityRight : Bool;   // Movement Executability
            movement164ExecutabilityLeft : Bool;   // Movement Executability
            movement164ExecutabilityRight : Bool;   // Movement Executability
            movement165ExecutabilityLeft : Bool;   // Movement Executability
            movement165ExecutabilityRight : Bool;   // Movement Executability
            movement166ExecutabilityLeft : Bool;   // Movement Executability
            movement166ExecutabilityRight : Bool;   // Movement Executability
            movement167ExecutabilityLeft : Bool;   // Movement Executability
            movement167ExecutabilityRight : Bool;   // Movement Executability
            movement168ExecutabilityLeft : Bool;   // Movement Executability
            movement168ExecutabilityRight : Bool;   // Movement Executability
            movement169ExecutabilityLeft : Bool;   // Movement Executability
            movement169ExecutabilityRight : Bool;   // Movement Executability
            movement170ExecutabilityLeft : Bool;   // Movement Executability
            movement170ExecutabilityRight : Bool;   // Movement Executability
            movement171ExecutabilityLeft : Bool;   // Movement Executability
            movement171ExecutabilityRight : Bool;   // Movement Executability
            movement172ExecutabilityLeft : Bool;   // Movement Executability
            movement172ExecutabilityRight : Bool;   // Movement Executability
            movement173ExecutabilityLeft : Bool;   // Movement Executability
            movement173ExecutabilityRight : Bool;   // Movement Executability
            movement174ExecutabilityLeft : Bool;   // Movement Executability
            movement174ExecutabilityRight : Bool;   // Movement Executability
            movement175ExecutabilityLeft : Bool;   // Movement Executability
            movement175ExecutabilityRight : Bool;   // Movement Executability
            movement176ExecutabilityLeft : Bool;   // Movement Executability
            movement176ExecutabilityRight : Bool;   // Movement Executability
            movement177ExecutabilityLeft : Bool;   // Movement Executability
            movement177ExecutabilityRight : Bool;   // Movement Executability
            movement178ExecutabilityLeft : Bool;   // Movement Executability
            movement178ExecutabilityRight : Bool;   // Movement Executability
            movement179ExecutabilityLeft : Bool;   // Movement Executability
            movement179ExecutabilityRight : Bool;   // Movement Executability
            movement180ExecutabilityLeft : Bool;   // Movement Executability
            movement180ExecutabilityRight : Bool;   // Movement Executability
            movement181ExecutabilityLeft : Bool;   // Movement Executability
            movement181ExecutabilityRight : Bool;   // Movement Executability
            movement182ExecutabilityLeft : Bool;   // Movement Executability
            movement182ExecutabilityRight : Bool;   // Movement Executability
            movement183ExecutabilityLeft : Bool;   // Movement Executability
            movement183ExecutabilityRight : Bool;   // Movement Executability
            movement184ExecutabilityLeft : Bool;   // Movement Executability
            movement184ExecutabilityRight : Bool;   // Movement Executability
            movement185ExecutabilityLeft : Bool;   // Movement Executability
            movement185ExecutabilityRight : Bool;   // Movement Executability
            movement186ExecutabilityLeft : Bool;   // Movement Executability
            movement186ExecutabilityRight : Bool;   // Movement Executability
            movement187ExecutabilityLeft : Bool;   // Movement Executability
            movement187ExecutabilityRight : Bool;   // Movement Executability
            movement188ExecutabilityLeft : Bool;   // Movement Executability
            movement188ExecutabilityRight : Bool;   // Movement Executability
            movement189ExecutabilityLeft : Bool;   // Movement Executability
            movement189ExecutabilityRight : Bool;   // Movement Executability
            movement190ExecutabilityLeft : Bool;   // Movement Executability
            movement190ExecutabilityRight : Bool;   // Movement Executability
            movement191ExecutabilityLeft : Bool;   // Movement Executability
            movement191ExecutabilityRight : Bool;   // Movement Executability
            movement192ExecutabilityLeft : Bool;   // Movement Executability
            movement192ExecutabilityRight : Bool;   // Movement Executability
            movement193ExecutabilityLeft : Bool;   // Movement Executability
            movement193ExecutabilityRight : Bool;   // Movement Executability
            movement194ExecutabilityLeft : Bool;   // Movement Executability
            movement194ExecutabilityRight : Bool;   // Movement Executability
            movement195ExecutabilityLeft : Bool;   // Movement Executability
            movement195ExecutabilityRight : Bool;   // Movement Executability
            movement196ExecutabilityLeft : Bool;   // Movement Executability
            movement196ExecutabilityRight : Bool;   // Movement Executability
            movement197ExecutabilityLeft : Bool;   // Movement Executability
            movement197ExecutabilityRight : Bool;   // Movement Executability
            movement198ExecutabilityLeft : Bool;   // Movement Executability
            movement198ExecutabilityRight : Bool;   // Movement Executability
            movement199ExecutabilityLeft : Bool;   // Movement Executability
            movement199ExecutabilityRight : Bool;   // Movement Executability
            movement200ExecutabilityLeft : Bool;   // Movement Executability
            movement200ExecutabilityRight : Bool;   // Movement Executability
            movement201ExecutabilityLeft : Bool;   // Movement Executability
            movement201ExecutabilityRight : Bool;   // Movement Executability
            movement202ExecutabilityLeft : Bool;   // Movement Executability
            movement202ExecutabilityRight : Bool;   // Movement Executability
            movement203ExecutabilityLeft : Bool;   // Movement Executability
            movement203ExecutabilityRight : Bool;   // Movement Executability
            movement204ExecutabilityLeft : Bool;   // Movement Executability
            movement204ExecutabilityRight : Bool;   // Movement Executability
            movement205ExecutabilityLeft : Bool;   // Movement Executability
            movement205ExecutabilityRight : Bool;   // Movement Executability
            movement206ExecutabilityLeft : Bool;   // Movement Executability
            movement206ExecutabilityRight : Bool;   // Movement Executability
            movement207ExecutabilityLeft : Bool;   // Movement Executability
            movement207ExecutabilityRight : Bool;   // Movement Executability
            movement208ExecutabilityLeft : Bool;   // Movement Executability
            movement208ExecutabilityRight : Bool;   // Movement Executability
            movement209ExecutabilityLeft : Bool;   // Movement Executability
            movement209ExecutabilityRight : Bool;   // Movement Executability
            movement210ExecutabilityLeft : Bool;   // Movement Executability
            movement210ExecutabilityRight : Bool;   // Movement Executability
            movement211ExecutabilityLeft : Bool;   // Movement Executability
            movement211ExecutabilityRight : Bool;   // Movement Executability
            movement212ExecutabilityLeft : Bool;   // Movement Executability
            movement212ExecutabilityRight : Bool;   // Movement Executability
            movement213ExecutabilityLeft : Bool;   // Movement Executability
            movement213ExecutabilityRight : Bool;   // Movement Executability
            movement214ExecutabilityLeft : Bool;   // Movement Executability
            movement214ExecutabilityRight : Bool;   // Movement Executability
            movement215ExecutabilityLeft : Bool;   // Movement Executability
            movement215ExecutabilityRight : Bool;   // Movement Executability
            movement216ExecutabilityLeft : Bool;   // Movement Executability
            movement216ExecutabilityRight : Bool;   // Movement Executability
            movement217ExecutabilityLeft : Bool;   // Movement Executability
            movement217ExecutabilityRight : Bool;   // Movement Executability
            movement218ExecutabilityLeft : Bool;   // Movement Executability
            movement218ExecutabilityRight : Bool;   // Movement Executability
            movement219ExecutabilityLeft : Bool;   // Movement Executability
            movement219ExecutabilityRight : Bool;   // Movement Executability
            movement220ExecutabilityLeft : Bool;   // Movement Executability
            movement220ExecutabilityRight : Bool;   // Movement Executability
            movement221ExecutabilityLeft : Bool;   // Movement Executability
            movement221ExecutabilityRight : Bool;   // Movement Executability
            movement222ExecutabilityLeft : Bool;   // Movement Executability
            movement222ExecutabilityRight : Bool;   // Movement Executability
            movement223ExecutabilityLeft : Bool;   // Movement Executability
            movement223ExecutabilityRight : Bool;   // Movement Executability
            movement224ExecutabilityLeft : Bool;   // Movement Executability
            movement224ExecutabilityRight : Bool;   // Movement Executability
            movement225ExecutabilityLeft : Bool;   // Movement Executability
            movement225ExecutabilityRight : Bool;   // Movement Executability
            movement226ExecutabilityLeft : Bool;   // Movement Executability
            movement226ExecutabilityRight : Bool;   // Movement Executability
            movement227ExecutabilityLeft : Bool;   // Movement Executability
            movement227ExecutabilityRight : Bool;   // Movement Executability
            movement228ExecutabilityLeft : Bool;   // Movement Executability
            movement228ExecutabilityRight : Bool;   // Movement Executability
            movement229ExecutabilityLeft : Bool;   // Movement Executability
            movement229ExecutabilityRight : Bool;   // Movement Executability
            movement230ExecutabilityLeft : Bool;   // Movement Executability
            movement230ExecutabilityRight : Bool;   // Movement Executability
            movement231ExecutabilityLeft : Bool;   // Movement Executability
            movement231ExecutabilityRight : Bool;   // Movement Executability
            movement232ExecutabilityLeft : Bool;   // Movement Executability
            movement232ExecutabilityRight : Bool;   // Movement Executability
            movement233ExecutabilityLeft : Bool;   // Movement Executability
            movement233ExecutabilityRight : Bool;   // Movement Executability
            movement234ExecutabilityLeft : Bool;   // Movement Executability
            movement234ExecutabilityRight : Bool;   // Movement Executability
            movement235ExecutabilityLeft : Bool;   // Movement Executability
            movement235ExecutabilityRight : Bool;   // Movement Executability
            movement236ExecutabilityLeft : Bool;   // Movement Executability
            movement236ExecutabilityRight : Bool;   // Movement Executability
            movement237ExecutabilityLeft : Bool;   // Movement Executability
            movement237ExecutabilityRight : Bool;   // Movement Executability
            movement238ExecutabilityLeft : Bool;   // Movement Executability
            movement238ExecutabilityRight : Bool;   // Movement Executability
            movement239ExecutabilityLeft : Bool;   // Movement Executability
            movement239ExecutabilityRight : Bool;   // Movement Executability
            movement240ExecutabilityLeft : Bool;   // Movement Executability
            movement240ExecutabilityRight : Bool;   // Movement Executability
            movement241ExecutabilityLeft : Bool;   // Movement Executability
            movement241ExecutabilityRight : Bool;   // Movement Executability
            movement242ExecutabilityLeft : Bool;   // Movement Executability
            movement242ExecutabilityRight : Bool;   // Movement Executability
            movement243ExecutabilityLeft : Bool;   // Movement Executability
            movement243ExecutabilityRight : Bool;   // Movement Executability
            movement244ExecutabilityLeft : Bool;   // Movement Executability
            movement244ExecutabilityRight : Bool;   // Movement Executability
            movement245ExecutabilityLeft : Bool;   // Movement Executability
            movement245ExecutabilityRight : Bool;   // Movement Executability
            movement246ExecutabilityLeft : Bool;   // Movement Executability
            movement246ExecutabilityRight : Bool;   // Movement Executability
            movement247ExecutabilityLeft : Bool;   // Movement Executability
            movement247ExecutabilityRight : Bool;   // Movement Executability
            movement248ExecutabilityLeft : Bool;   // Movement Executability
            movement248ExecutabilityRight : Bool;   // Movement Executability
            movement249ExecutabilityLeft : Bool;   // Movement Executability
            movement249ExecutabilityRight : Bool;   // Movement Executability
            movement250ExecutabilityLeft : Bool;   // Movement Executability
            movement250ExecutabilityRight : Bool;   // Movement Executability
            movement251ExecutabilityLeft : Bool;   // Movement Executability
            movement251ExecutabilityRight : Bool;   // Movement Executability
            movement252ExecutabilityLeft : Bool;   // Movement Executability
            movement252ExecutabilityRight : Bool;   // Movement Executability
            movement253ExecutabilityLeft : Bool;   // Movement Executability
            movement253ExecutabilityRight : Bool;   // Movement Executability
            movement254ExecutabilityLeft : Bool;   // Movement Executability
            movement254ExecutabilityRight : Bool;   // Movement Executability
            movement255ExecutabilityLeft : Bool;   // Movement Executability
            movement255ExecutabilityRight : Bool;   // Movement Executability
            movement256ExecutabilityLeft : Bool;   // Movement Executability
            movement256ExecutabilityRight : Bool;   // Movement Executability
         END_STRUCT;
         MovementActive : Struct   // Movement Active
            movement1ActiveLeft : Bool;   // Movement Active
            movement1ActiveRight : Bool;   // Movement Active
            movement2ActiveLeft : Bool;   // Movement Active
            movement2ActiveRight : Bool;   // Movement Active
            movement3ActiveLeft : Bool;   // Movement Active
            movement3ActiveRight : Bool;   // Movement Active
            movement4ActiveLeft : Bool;   // Movement Active
            movement4ActiveRight : Bool;   // Movement Active
            movement5ActiveLeft : Bool;   // Movement Active
            movement5ActiveRight : Bool;   // Movement Active
            movement6ActiveLeft : Bool;   // Movement Active
            movement6ActiveRight : Bool;   // Movement Active
            movement7ActiveLeft : Bool;   // Movement Active
            movement7ActiveRight : Bool;   // Movement Active
            movement8ActiveLeft : Bool;   // Movement Active
            movement8ActiveRight : Bool;   // Movement Active
            movement9ActiveLeft : Bool;   // Movement Active
            movement9ActiveRight : Bool;   // Movement Active
            movement10ActiveLeft : Bool;   // Movement Active
            movement10ActiveRight : Bool;   // Movement Active
            movement11ActiveLeft : Bool;   // Movement Active
            movement11ActiveRight : Bool;   // Movement Active
            movement12ActiveLeft : Bool;   // Movement Active
            movement12ActiveRight : Bool;   // Movement Active
            movement13ActiveLeft : Bool;   // Movement Active
            movement13ActiveRight : Bool;   // Movement Active
            movement14ActiveLeft : Bool;   // Movement Active
            movement14ActiveRight : Bool;   // Movement Active
            movement15ActiveLeft : Bool;   // Movement Active
            movement15ActiveRight : Bool;   // Movement Active
            movement16ActiveLeft : Bool;   // Movement Active
            movement16ActiveRight : Bool;   // Movement Active
            movement17ActiveLeft : Bool;   // Movement Active
            movement17ActiveRight : Bool;   // Movement Active
            movement18ActiveLeft : Bool;   // Movement Active
            movement18ActiveRight : Bool;   // Movement Active
            movement19ActiveLeft : Bool;   // Movement Active
            movement19ActiveRight : Bool;   // Movement Active
            movement20ActiveLeft : Bool;   // Movement Active
            movement20ActiveRight : Bool;   // Movement Active
            movement21ActiveLeft : Bool;   // Movement Active
            movement21ActiveRight : Bool;   // Movement Active
            movement22ActiveLeft : Bool;   // Movement Active
            movement22ActiveRight : Bool;   // Movement Active
            movement23ActiveLeft : Bool;   // Movement Active
            movement23ActiveRight : Bool;   // Movement Active
            movement24ActiveLeft : Bool;   // Movement Active
            movement24ActiveRight : Bool;   // Movement Active
            movement25ActiveLeft : Bool;   // Movement Active
            movement25ActiveRight : Bool;   // Movement Active
            movement26ActiveLeft : Bool;   // Movement Active
            movement26ActiveRight : Bool;   // Movement Active
            movement27ActiveLeft : Bool;   // Movement Active
            movement27ActiveRight : Bool;   // Movement Active
            movement28ActiveLeft : Bool;   // Movement Active
            movement28ActiveRight : Bool;   // Movement Active
            movement29ActiveLeft : Bool;   // Movement Active
            movement29ActiveRight : Bool;   // Movement Active
            movement30ActiveLeft : Bool;   // Movement Active
            movement30ActiveRight : Bool;   // Movement Active
            movement31ActiveLeft : Bool;   // Movement Active
            movement31ActiveRight : Bool;   // Movement Active
            movement32ActiveLeft : Bool;   // Movement Active
            movement32ActiveRight : Bool;   // Movement Active
            movement33ActiveLeft : Bool;   // Movement Active
            movement33ActiveRight : Bool;   // Movement Active
            movement34ActiveLeft : Bool;   // Movement Active
            movement34ActiveRight : Bool;   // Movement Active
            movement35ActiveLeft : Bool;   // Movement Active
            movement35ActiveRight : Bool;   // Movement Active
            movement36ActiveLeft : Bool;   // Movement Active
            movement36ActiveRight : Bool;   // Movement Active
            movement37ActiveLeft : Bool;   // Movement Active
            movement37ActiveRight : Bool;   // Movement Active
            movement38ActiveLeft : Bool;   // Movement Active
            movement38ActiveRight : Bool;   // Movement Active
            movement39ActiveLeft : Bool;   // Movement Active
            movement39ActiveRight : Bool;   // Movement Active
            movement40ActiveLeft : Bool;   // Movement Active
            movement40ActiveRight : Bool;   // Movement Active
            movement41ActiveLeft : Bool;   // Movement Active
            movement41ActiveRight : Bool;   // Movement Active
            movement42ActiveLeft : Bool;   // Movement Active
            movement42ActiveRight : Bool;   // Movement Active
            movement43ActiveLeft : Bool;   // Movement Active
            movement43ActiveRight : Bool;   // Movement Active
            movement44ActiveLeft : Bool;   // Movement Active
            movement44ActiveRight : Bool;   // Movement Active
            movement45ActiveLeft : Bool;   // Movement Active
            movement45ActiveRight : Bool;   // Movement Active
            movement46ActiveLeft : Bool;   // Movement Active
            movement46ActiveRight : Bool;   // Movement Active
            movement47ActiveLeft : Bool;   // Movement Active
            movement47ActiveRight : Bool;   // Movement Active
            movement48ActiveLeft : Bool;   // Movement Active
            movement48ActiveRight : Bool;   // Movement Active
            movement49ActiveLeft : Bool;   // Movement Active
            movement49ActiveRight : Bool;   // Movement Active
            movement50ActiveLeft : Bool;   // Movement Active
            movement50ActiveRight : Bool;   // Movement Active
            movement51ActiveLeft : Bool;   // Movement Active
            movement51ActiveRight : Bool;   // Movement Active
            movement52ActiveLeft : Bool;   // Movement Active
            movement52ActiveRight : Bool;   // Movement Active
            movement53ActiveLeft : Bool;   // Movement Active
            movement53ActiveRight : Bool;   // Movement Active
            movement54ActiveLeft : Bool;   // Movement Active
            movement54ActiveRight : Bool;   // Movement Active
            movement55ActiveLeft : Bool;   // Movement Active
            movement55ActiveRight : Bool;   // Movement Active
            movement56ActiveLeft : Bool;   // Movement Active
            movement56ActiveRight : Bool;   // Movement Active
            movement57ActiveLeft : Bool;   // Movement Active
            movement57ActiveRight : Bool;   // Movement Active
            movement58ActiveLeft : Bool;   // Movement Active
            movement58ActiveRight : Bool;   // Movement Active
            movement59ActiveLeft : Bool;   // Movement Active
            movement59ActiveRight : Bool;   // Movement Active
            movement60ActiveLeft : Bool;   // Movement Active
            movement60ActiveRight : Bool;   // Movement Active
            movement61ActiveLeft : Bool;   // Movement Active
            movement61ActiveRight : Bool;   // Movement Active
            movement62ActiveLeft : Bool;   // Movement Active
            movement62ActiveRight : Bool;   // Movement Active
            movement63ActiveLeft : Bool;   // Movement Active
            movement63ActiveRight : Bool;   // Movement Active
            movement64ActiveLeft : Bool;   // Movement Active
            movement64ActiveRight : Bool;   // Movement Active
            movement65ActiveLeft : Bool;   // Movement Active
            movement65ActiveRight : Bool;   // Movement Active
            movement66ActiveLeft : Bool;   // Movement Active
            movement66ActiveRight : Bool;   // Movement Active
            movement67ActiveLeft : Bool;   // Movement Active
            movement67ActiveRight : Bool;   // Movement Active
            movement68ActiveLeft : Bool;   // Movement Active
            movement68ActiveRight : Bool;   // Movement Active
            movement69ActiveLeft : Bool;   // Movement Active
            movement69ActiveRight : Bool;   // Movement Active
            movement70ActiveLeft : Bool;   // Movement Active
            movement70ActiveRight : Bool;   // Movement Active
            movement71ActiveLeft : Bool;   // Movement Active
            movement71ActiveRight : Bool;   // Movement Active
            movement72ActiveLeft : Bool;   // Movement Active
            movement72ActiveRight : Bool;   // Movement Active
            movement73ActiveLeft : Bool;   // Movement Active
            movement73ActiveRight : Bool;   // Movement Active
            movement74ActiveLeft : Bool;   // Movement Active
            movement74ActiveRight : Bool;   // Movement Active
            movement75ActiveLeft : Bool;   // Movement Active
            movement75ActiveRight : Bool;   // Movement Active
            movement76ActiveLeft : Bool;   // Movement Active
            movement76ActiveRight : Bool;   // Movement Active
            movement77ActiveLeft : Bool;   // Movement Active
            movement77ActiveRight : Bool;   // Movement Active
            movement78ActiveLeft : Bool;   // Movement Active
            movement78ActiveRight : Bool;   // Movement Active
            movement79ActiveLeft : Bool;   // Movement Active
            movement79ActiveRight : Bool;   // Movement Active
            movement80ActiveLeft : Bool;   // Movement Active
            movement80ActiveRight : Bool;   // Movement Active
            movement81ActiveLeft : Bool;   // Movement Active
            movement81ActiveRight : Bool;   // Movement Active
            movement82ActiveLeft : Bool;   // Movement Active
            movement82ActiveRight : Bool;   // Movement Active
            movement83ActiveLeft : Bool;   // Movement Active
            movement83ActiveRight : Bool;   // Movement Active
            movement84ActiveLeft : Bool;   // Movement Active
            movement84ActiveRight : Bool;   // Movement Active
            movement85ActiveLeft : Bool;   // Movement Active
            movement85ActiveRight : Bool;   // Movement Active
            movement86ActiveLeft : Bool;   // Movement Active
            movement86ActiveRight : Bool;   // Movement Active
            movement87ActiveLeft : Bool;   // Movement Active
            movement87ActiveRight : Bool;   // Movement Active
            movement88ActiveLeft : Bool;   // Movement Active
            movement88ActiveRight : Bool;   // Movement Active
            movement89ActiveLeft : Bool;   // Movement Active
            movement89ActiveRight : Bool;   // Movement Active
            movement90ActiveLeft : Bool;   // Movement Active
            movement90ActiveRight : Bool;   // Movement Active
            movement91ActiveLeft : Bool;   // Movement Active
            movement91ActiveRight : Bool;   // Movement Active
            movement92ActiveLeft : Bool;   // Movement Active
            movement92ActiveRight : Bool;   // Movement Active
            movement93ActiveLeft : Bool;   // Movement Active
            movement93ActiveRight : Bool;   // Movement Active
            movement94ActiveLeft : Bool;   // Movement Active
            movement94ActiveRight : Bool;   // Movement Active
            movement95ActiveLeft : Bool;   // Movement Active
            movement95ActiveRight : Bool;   // Movement Active
            movement96ActiveLeft : Bool;   // Movement Active
            movement96ActiveRight : Bool;   // Movement Active
            movement97ActiveLeft : Bool;   // Movement Active
            movement97ActiveRight : Bool;   // Movement Active
            movement98ActiveLeft : Bool;   // Movement Active
            movement98ActiveRight : Bool;   // Movement Active
            movement99ActiveLeft : Bool;   // Movement Active
            movement99ActiveRight : Bool;   // Movement Active
            movement100ActiveLeft : Bool;   // Movement Active
            movement100ActiveRight : Bool;   // Movement Active
            movement101ActiveLeft : Bool;   // Movement Active
            movement101ActiveRight : Bool;   // Movement Active
            movement102ActiveLeft : Bool;   // Movement Active
            movement102ActiveRight : Bool;   // Movement Active
            movement103ActiveLeft : Bool;   // Movement Active
            movement103ActiveRight : Bool;   // Movement Active
            movement104ActiveLeft : Bool;   // Movement Active
            movement104ActiveRight : Bool;   // Movement Active
            movement105ActiveLeft : Bool;   // Movement Active
            movement105ActiveRight : Bool;   // Movement Active
            movement106ActiveLeft : Bool;   // Movement Active
            movement106ActiveRight : Bool;   // Movement Active
            movement107ActiveLeft : Bool;   // Movement Active
            movement107ActiveRight : Bool;   // Movement Active
            movement108ActiveLeft : Bool;   // Movement Active
            movement108ActiveRight : Bool;   // Movement Active
            movement109ActiveLeft : Bool;   // Movement Active
            movement109ActiveRight : Bool;   // Movement Active
            movement110ActiveLeft : Bool;   // Movement Active
            movement110ActiveRight : Bool;   // Movement Active
            movement111ActiveLeft : Bool;   // Movement Active
            movement111ActiveRight : Bool;   // Movement Active
            movement112ActiveLeft : Bool;   // Movement Active
            movement112ActiveRight : Bool;   // Movement Active
            movement113ActiveLeft : Bool;   // Movement Active
            movement113ActiveRight : Bool;   // Movement Active
            movement114ActiveLeft : Bool;   // Movement Active
            movement114ActiveRight : Bool;   // Movement Active
            movement115ActiveLeft : Bool;   // Movement Active
            movement115ActiveRight : Bool;   // Movement Active
            movement116ActiveLeft : Bool;   // Movement Active
            movement116ActiveRight : Bool;   // Movement Active
            movement117ActiveLeft : Bool;   // Movement Active
            movement117ActiveRight : Bool;   // Movement Active
            movement118ActiveLeft : Bool;   // Movement Active
            movement118ActiveRight : Bool;   // Movement Active
            movement119ActiveLeft : Bool;   // Movement Active
            movement119ActiveRight : Bool;   // Movement Active
            movement120ActiveLeft : Bool;   // Movement Active
            movement120ActiveRight : Bool;   // Movement Active
            movement121ActiveLeft : Bool;   // Movement Active
            movement121ActiveRight : Bool;   // Movement Active
            movement122ActiveLeft : Bool;   // Movement Active
            movement122ActiveRight : Bool;   // Movement Active
            movement123ActiveLeft : Bool;   // Movement Active
            movement123ActiveRight : Bool;   // Movement Active
            movement124ActiveLeft : Bool;   // Movement Active
            movement124ActiveRight : Bool;   // Movement Active
            movement125ActiveLeft : Bool;   // Movement Active
            movement125ActiveRight : Bool;   // Movement Active
            movement126ActiveLeft : Bool;   // Movement Active
            movement126ActiveRight : Bool;   // Movement Active
            movement127ActiveLeft : Bool;   // Movement Active
            movement127ActiveRight : Bool;   // Movement Active
            movement128ActiveLeft : Bool;   // Movement Active
            movement128ActiveRight : Bool;   // Movement Active
            movement129ActiveLeft : Bool;   // Movement Active
            movement129ActiveRight : Bool;   // Movement Active
            movement130ActiveLeft : Bool;   // Movement Active
            movement130ActiveRight : Bool;   // Movement Active
            movement131ActiveLeft : Bool;   // Movement Active
            movement131ActiveRight : Bool;   // Movement Active
            movement132ActiveLeft : Bool;   // Movement Active
            movement132ActiveRight : Bool;   // Movement Active
            movement133ActiveLeft : Bool;   // Movement Active
            movement133ActiveRight : Bool;   // Movement Active
            movement134ActiveLeft : Bool;   // Movement Active
            movement134ActiveRight : Bool;   // Movement Active
            movement135ActiveLeft : Bool;   // Movement Active
            movement135ActiveRight : Bool;   // Movement Active
            movement136ActiveLeft : Bool;   // Movement Active
            movement136ActiveRight : Bool;   // Movement Active
            movement137ActiveLeft : Bool;   // Movement Active
            movement137ActiveRight : Bool;   // Movement Active
            movement138ActiveLeft : Bool;   // Movement Active
            movement138ActiveRight : Bool;   // Movement Active
            movement139ActiveLeft : Bool;   // Movement Active
            movement139ActiveRight : Bool;   // Movement Active
            movement140ActiveLeft : Bool;   // Movement Active
            movement140ActiveRight : Bool;   // Movement Active
            movement141ActiveLeft : Bool;   // Movement Active
            movement141ActiveRight : Bool;   // Movement Active
            movement142ActiveLeft : Bool;   // Movement Active
            movement142ActiveRight : Bool;   // Movement Active
            movement143ActiveLeft : Bool;   // Movement Active
            movement143ActiveRight : Bool;   // Movement Active
            movement144ActiveLeft : Bool;   // Movement Active
            movement144ActiveRight : Bool;   // Movement Active
            movement145ActiveLeft : Bool;   // Movement Active
            movement145ActiveRight : Bool;   // Movement Active
            movement146ActiveLeft : Bool;   // Movement Active
            movement146ActiveRight : Bool;   // Movement Active
            movement147ActiveLeft : Bool;   // Movement Active
            movement147ActiveRight : Bool;   // Movement Active
            movement148ActiveLeft : Bool;   // Movement Active
            movement148ActiveRight : Bool;   // Movement Active
            movement149ActiveLeft : Bool;   // Movement Active
            movement149ActiveRight : Bool;   // Movement Active
            movement150ActiveLeft : Bool;   // Movement Active
            movement150ActiveRight : Bool;   // Movement Active
            movement151ActiveLeft : Bool;   // Movement Active
            movement151ActiveRight : Bool;   // Movement Active
            movement152ActiveLeft : Bool;   // Movement Active
            movement152ActiveRight : Bool;   // Movement Active
            movement153ActiveLeft : Bool;   // Movement Active
            movement153ActiveRight : Bool;   // Movement Active
            movement154ActiveLeft : Bool;   // Movement Active
            movement154ActiveRight : Bool;   // Movement Active
            movement155ActiveLeft : Bool;   // Movement Active
            movement155ActiveRight : Bool;   // Movement Active
            movement156ActiveLeft : Bool;   // Movement Active
            movement156ActiveRight : Bool;   // Movement Active
            movement157ActiveLeft : Bool;   // Movement Active
            movement157ActiveRight : Bool;   // Movement Active
            movement158ActiveLeft : Bool;   // Movement Active
            movement158ActiveRight : Bool;   // Movement Active
            movement159ActiveLeft : Bool;   // Movement Active
            movement159ActiveRight : Bool;   // Movement Active
            movement160ActiveLeft : Bool;   // Movement Active
            movement160ActiveRight : Bool;   // Movement Active
            movement161ActiveLeft : Bool;   // Movement Active
            movement161ActiveRight : Bool;   // Movement Active
            movement162ActiveLeft : Bool;   // Movement Active
            movement162ActiveRight : Bool;   // Movement Active
            movement163ActiveLeft : Bool;   // Movement Active
            movement163ActiveRight : Bool;   // Movement Active
            movement164ActiveLeft : Bool;   // Movement Active
            movement164ActiveRight : Bool;   // Movement Active
            movement165ActiveLeft : Bool;   // Movement Active
            movement165ActiveRight : Bool;   // Movement Active
            movement166ActiveLeft : Bool;   // Movement Active
            movement166ActiveRight : Bool;   // Movement Active
            movement167ActiveLeft : Bool;   // Movement Active
            movement167ActiveRight : Bool;   // Movement Active
            movement168ActiveLeft : Bool;   // Movement Active
            movement168ActiveRight : Bool;   // Movement Active
            movement169ActiveLeft : Bool;   // Movement Active
            movement169ActiveRight : Bool;   // Movement Active
            movement170ActiveLeft : Bool;   // Movement Active
            movement170ActiveRight : Bool;   // Movement Active
            movement171ActiveLeft : Bool;   // Movement Active
            movement171ActiveRight : Bool;   // Movement Active
            movement172ActiveLeft : Bool;   // Movement Active
            movement172ActiveRight : Bool;   // Movement Active
            movement173ActiveLeft : Bool;   // Movement Active
            movement173ActiveRight : Bool;   // Movement Active
            movement174ActiveLeft : Bool;   // Movement Active
            movement174ActiveRight : Bool;   // Movement Active
            movement175ActiveLeft : Bool;   // Movement Active
            movement175ActiveRight : Bool;   // Movement Active
            movement176ActiveLeft : Bool;   // Movement Active
            movement176ActiveRight : Bool;   // Movement Active
            movement177ActiveLeft : Bool;   // Movement Active
            movement177ActiveRight : Bool;   // Movement Active
            movement178ActiveLeft : Bool;   // Movement Active
            movement178ActiveRight : Bool;   // Movement Active
            movement179ActiveLeft : Bool;   // Movement Active
            movement179ActiveRight : Bool;   // Movement Active
            movement180ActiveLeft : Bool;   // Movement Active
            movement180ActiveRight : Bool;   // Movement Active
            movement181ActiveLeft : Bool;   // Movement Active
            movement181ActiveRight : Bool;   // Movement Active
            movement182ActiveLeft : Bool;   // Movement Active
            movement182ActiveRight : Bool;   // Movement Active
            movement183ActiveLeft : Bool;   // Movement Active
            movement183ActiveRight : Bool;   // Movement Active
            movement184ActiveLeft : Bool;   // Movement Active
            movement184ActiveRight : Bool;   // Movement Active
            movement185ActiveLeft : Bool;   // Movement Active
            movement185ActiveRight : Bool;   // Movement Active
            movement186ActiveLeft : Bool;   // Movement Active
            movement186ActiveRight : Bool;   // Movement Active
            movement187ActiveLeft : Bool;   // Movement Active
            movement187ActiveRight : Bool;   // Movement Active
            movement188ActiveLeft : Bool;   // Movement Active
            movement188ActiveRight : Bool;   // Movement Active
            movement189ActiveLeft : Bool;   // Movement Active
            movement189ActiveRight : Bool;   // Movement Active
            movement190ActiveLeft : Bool;   // Movement Active
            movement190ActiveRight : Bool;   // Movement Active
            movement191ActiveLeft : Bool;   // Movement Active
            movement191ActiveRight : Bool;   // Movement Active
            movement192ActiveLeft : Bool;   // Movement Active
            movement192ActiveRight : Bool;   // Movement Active
            movement193ActiveLeft : Bool;   // Movement Active
            movement193ActiveRight : Bool;   // Movement Active
            movement194ActiveLeft : Bool;   // Movement Active
            movement194ActiveRight : Bool;   // Movement Active
            movement195ActiveLeft : Bool;   // Movement Active
            movement195ActiveRight : Bool;   // Movement Active
            movement196ActiveLeft : Bool;   // Movement Active
            movement196ActiveRight : Bool;   // Movement Active
            movement197ActiveLeft : Bool;   // Movement Active
            movement197ActiveRight : Bool;   // Movement Active
            movement198ActiveLeft : Bool;   // Movement Active
            movement198ActiveRight : Bool;   // Movement Active
            movement199ActiveLeft : Bool;   // Movement Active
            movement199ActiveRight : Bool;   // Movement Active
            movement200ActiveLeft : Bool;   // Movement Active
            movement200ActiveRight : Bool;   // Movement Active
            movement201ActiveLeft : Bool;   // Movement Active
            movement201ActiveRight : Bool;   // Movement Active
            movement202ActiveLeft : Bool;   // Movement Active
            movement202ActiveRight : Bool;   // Movement Active
            movement203ActiveLeft : Bool;   // Movement Active
            movement203ActiveRight : Bool;   // Movement Active
            movement204ActiveLeft : Bool;   // Movement Active
            movement204ActiveRight : Bool;   // Movement Active
            movement205ActiveLeft : Bool;   // Movement Active
            movement205ActiveRight : Bool;   // Movement Active
            movement206ActiveLeft : Bool;   // Movement Active
            movement206ActiveRight : Bool;   // Movement Active
            movement207ActiveLeft : Bool;   // Movement Active
            movement207ActiveRight : Bool;   // Movement Active
            movement208ActiveLeft : Bool;   // Movement Active
            movement208ActiveRight : Bool;   // Movement Active
            movement209ActiveLeft : Bool;   // Movement Active
